// TIA Portal V20 export
DATA_BLOCK "ControlNodes"   // DB32
// stored: MemoryReserve 100, Namespace Unit1
   VAR
      em { ExternalWritable := 'False'} : "LAF_typeEmControlNode";
      fuse : Array[0..150] of Bool;
      pws : Array[0..10] of Bool;
      motorPowerMC { ExternalWritable := 'False'} : Struct
         FeedBack : Bool;
         mcOn : Bool;
         Ready : Bool;
         Operation : Bool;
         Run : Bool;
         Fault : Bool;
         Error : Bool;
      END_STRUCT;
      airOK { ExternalWritable := 'False'} : Bool;   // Compressed air OK
      InitializeEnable { ExternalWritable := 'False'} : Bool;
      AutoStartEnable { ExternalWritable := 'False'} : Bool;
      cmFFU_LIU117 : "LER_typeLIU117ControlNode";
      citiMap : "LER_OEM_Data";
      "========Communication========" : Bool;
      BA030 { ExternalWritable := 'False'} : "LER_typeCommunicationControlNode";
      BA040 { ExternalWritable := 'False'} : "LER_typeCommunicationControlNode";
      BA100 { S7_SetPoint := 'True'} : "LER_typeCommunicationControlNode";
      ConveyorA { ExternalWritable := 'False'} : "LER_typeCommunicationControlNode";
   END_VAR
BEGIN
   // fuse[0] : KISTLER 100KN PRESS POWER TRIPPED E202CB
   // fuse[1] : KISTLER 100KN PRESS POWER TRIPPED E208CB
   // fuse[2] : KISTLER 30KN PRESS POWER TRIPPED E214CB
   // fuse[3] : SPARE
   // fuse[4] : SPARE
   // fuse[5] : E8404PWS CONTROLLER POWER SMPS AC POWER TRIPPED E320CB
   // fuse[6] : E8704PWS SAFETY POWER SMPS AC POWER TRIPPED E326CB
   // fuse[7] : E8804PWS CONTRL POWER SMPS AC POWER TRIPPED E332CB
   // fuse[8] : PROCESSOR POWER ON TIPPRED E4120CB
   // fuse[9] : PROGRAMING POWER OUTLET TRPPED E4126CB
   // fuse[10] : SPARE
   // fuse[11] : PANEL LED POWER TRIPPED E4304CB
   // fuse[12] : SPARE
   // fuse[13] : CONTROL LEVEL HUB POWER TRIPPED E4420CB
   // fuse[14] : MAIN HMI POWER TRIPPED E4426CB
   // fuse[15] : PORTABLE HMI POWER TIPPED E4432CB
   // fuse[16] : PORTABLE HMI POWER TIPPED E4456CB
   // fuse[17] : 120VAC HEATER-1 POWER TR PRIMARY TRIPPED E5100CB
   // fuse[18] : SPARE
   // fuse[19] : SPARE
   // fuse[20] : UPPER 1-1 HEATER POWER TRIPPED E5156CB
   // fuse[21] : UPPER 1-2 HEATER POWER TRIPPED E5162CB
   // fuse[22] : LOWER 1-1 HEATER POWER TRIPPED E5168CB
   // fuse[23] : LOWER 1-2 HEATER POWER TRIPPED E5174CB
   // fuse[24] : LOWER 1-3 HEATER POWER TRIPPED E5180CB
   // fuse[25] : SPARE
   // fuse[26] : 120VAC HEATER-2 POWER TR PRIMARY TRIPPED E6100CB
   // fuse[27] : SPARE
   // fuse[28] : SPARE
   // fuse[29] : UPPER 2-1 HEATER POWER TRIPPED E6156CB
   // fuse[30] : UPPER 2-2 HEATER POWER TRIPPED E6162CB
   // fuse[31] : LOWER 2-1 HEATER POWER TRIPPED E6168CB
   // fuse[32] : LOWER 2-2 HEATER POWER TRIPPED E6174CB
   // fuse[33] : LOWER 2-3 HEATER POWER TRIPPED E6180CB
   // fuse[34] : SPARE
   // fuse[35] : 120VAC CONTROL POWER TR PRIMARY TRIPPED E7100CB
   // fuse[36] : 120VAC CONTROL POWER TR SECONDARY TRIPPED E7110CB
   // fuse[37] : CONTROL POWER ON TRIPPED E7116CB
   // fuse[38] : MOTOR PANEL CONTROL POWER TRIPPED E7154CB
   // fuse[39] : POWER STRIP OUTLET POWER TRIPPED E7160CB
   // fuse[40] : POWER STRIP OUTLET POWER TRIPPED E7166CB
   // fuse[41] : QR LASER MARKING TRIPPED E7172CB
   // fuse[42] : HI-POT TESTER POWER TRIPPED E7178CB
   // fuse[43] : FFU-1 POWER TRIPPED E7222CB
   // fuse[44] : UPPER 1-1 TEMPERATURE CONTROLLER POWER TRIPPED E5206CB
   // fuse[45] : UPPER 1-2 TEMPERATURE CONTROLLER POWER TRIPPED E5212CB
   // fuse[46] : LOWER 1-1 TEMPERATURE CONTROLLER POWER TRIPPED E5218CB
   // fuse[47] : LOWER 1-2 TEMPERATURE CONTROLLER POWER TRIPPED E5224CB
   // fuse[48] : LOWER 1-3 TEMPERATURE CONTROLLER POWER TRIPPED E5230CB
   // fuse[49] : UPPER 2-1 TEMPERATURE CONTROLLER POWER TRIPPED E6206CB
   // fuse[50] : UPPER 2-2 TEMPERATURE CONTROLLER POWER TRIPPED E6212CB
   // fuse[51] : LOWER 2-1 TEMPERATURE CONTROLLER POWER TRIPPED E6218CB
   // fuse[52] : LOWER 2-2 TEMPERATURE CONTROLLER POWER TRIPPED E6224CB
   // fuse[53] : LOWER 2-3 TEMPERATURE CONTROLLER POWER TRIPPED E6230CB
   // fuse[54] : SPARE
   // fuse[55] : ET200MP I/O OUTPUT POWER TRIPPED E8154CB
   // fuse[56] : JUNCTION BOX CONTROL POWER TRIPPED E8180CB
   // fuse[57] : CLASS 2 SMPS POWER TRIPPED E8204CB
   // fuse[58] : ET200ECO PN-1 POWER TRIPPED E8220CB
   // fuse[59] : ET200ECO PN-2 POWER TRIPPED E8224CB
   // fuse[60] : ET200ECO PN-3 POWER TRIPPED E8228CB
   // fuse[61] : ET200ECO PN-4 POWER TRIPPED E8232CB
   // fuse[62] : PANEL FAN POWER TRIPPED E8304CB
   // fuse[63] : SPARE
   // fuse[64] : CONTROLLER DC POWER TRIPPED E8406CB
   // fuse[65] : KISTLER CONTROL POWER TRIPPED E8416CB
   // fuse[66] : MANIFOLD-1 POWER TRIPPED E8422CB
   // fuse[67] : MANIFOLD-2 POWER TRIPPED E8430CB
   // fuse[68] : QR READER POWER TRIPPED E8456CB
   // fuse[69] : QR READER POWER TRIPPED E8462CB
   // fuse[70] : HANDY QR READER POWER TRIPPED E8468CB
   // fuse[71] : PROFINET CONVERTER POWER TRIPPED E8474CB
   // fuse[72] : MONITORING RELAY POWER TRIPPED E8504CB
   // fuse[73] : SPARE
   // fuse[74] : SAFETY DC POWER TRIPPED E8706CB
   // fuse[75] : ET200SP I/O SAFETY POWER TRIPPED E8716CB
   // fuse[76] : JUNCTION BOX CONTROL POWER TRIPPED E8736CB
   // fuse[77] : ET200ECO PN SAFETYT-1 POWER TRIPPED E8756CB
   // fuse[78] : ET200ECO PN SAFETYT-2 POWER TRIPPED E8762CB
   // fuse[79] : SPARE
   // fuse[80] : CONTROL DC POWER TRIPPED E8806CB
   // fuse[81] : JUNCTION BOX CONTROL POWER TRIPPED E8816CB
   // fuse[82] : DRIVE-CLIQ HUB POWER TRIPPED E8822CB
   // fuse[83] : EQUIPMENT LED POWER TRIPPED E8828CB
   // fuse[84] : SPARE
   // fuse[85] : SAFETY DC POWER TRIPPED E218CB
   // fuse[86] : CLASS 2 SMPS POWER TRIPPED E308CB
   // fuse[87] : ET200ECO PN-1 POWER TRIPPED E324CB
   // fuse[88] : ET200ECO PN-2 POWER TRIPPED E328CB
   // fuse[89] : ET200ECO PN-3 POWER TRIPPED E332CB
   // fuse[90] : ET200ECO PN-4 POWER TRIPPED E336CB
   // fuse[91] : MOTOR POWER MC FEEDBACK
   // fuse[92] : MOTOR POWER TRIPPED E202CB
   // fuse[93] : MAIN CONTROL PANEL MAIN POWER TRIPPED E208CB
   // fuse[94] : E6104PWS CONTROL POWER SMPS AC POWER TRIPPED E314CB
   // fuse[95] : JROUT P&P Y-AXIS POWER TR PRIMARY TRIPPED E400CB
   // fuse[96] : JROUT P&P Y-AXIS POWER TR ECONDARY TRIPPED E410CB
   // fuse[97] : INS PROCESS P&P X-AXIS POWER TR PRIMARY TRIPPED E500CB
   // fuse[98] : INS PROCESS P&P X-AXIS POWER TR ECONDARY TRIPPED E510CB
   // fuse[99] : JR UNLOADING Y-AXIS POWER TR PRIMARY TRIPPED E600CB
   // fuse[100] : JR UNLOADING Y-AXIS POWER TR ECONDARY TRIPPED E610CB
   // fuse[101] : POWER METER POWER TRIIPED E720CB
   // fuse[102] : POWER METER CONTROL POWER TRIIPED E726CB
   // fuse[103] : JR OUT P&P 1 Y-AXIS POWER ON TRIPPED E2004CB
   // fuse[104] : JR OUT P&P 2 Y-AXIS POWER ON TRIPPED E2104CB
   // fuse[105] : INS PROCESS P&P 1 X-AXIS POWER ON TRIPPED E2204CB
   // fuse[106] : INS PROCESS P&P 2 X-AXIS POWER ON TRIPPED E2304CB
   // fuse[107] : JR UNLOADING Y-AXIS POWER ON TRIPPED E2404CB
   // fuse[108] : MOTOR POWER MC COIL POWER TRIPPED E6156CB
   // fuse[109] : PROCESSOR POWER ON TRIPPRED E4116CB
   // fuse[110] : MAIN CONTROL PANEL HOT POWER TRIPPED E4156CB
   // fuse[111] : SYSTEM LEVEL HUB POWER TRIPPED E4162CB
   // fuse[112] : PANEL LED POWER TRIPPED E4304CB
   // fuse[113] : CONTROL POWER TRIPPED E5110CB
   // fuse[114] : CONTROL POWER ON TRIPPED E5120CB
   // fuse[115] : SERVON CONTROL POWER TRIPPED E6122CB
   // fuse[116] : SERVO CONTROL UNIT CONTROL POWER TRIPPED E6128CB
   // fuse[117] : PANEL FAN POWER TRIPPED E6204CB
   // fuse[118] : SPARE
   // fuse[119] : SPARE
   // fuse[120] : SPARE
   // fuse[121] : SPARE
   // pws[0] : PLC POWER SMPS DC OK E4404PWS
   // pws[1] : CONTROL POWER SMPS DC OK E8104PWS
   // pws[2] : CLASS 2 SMPS MONITORING E8206PWS
   // pws[3] : CONTROLLER POWER SMPS DC OK E8404PWS
   // pws[4] : SAFETY POWER SMPS DC OK E8704PWS
   // pws[5] : COONTRL POWER SMPS DC OK E8804PWS
   // pws[6] : CLASS 2 SMPS MONITORING E310PWS
   // pws[7] : CONTROL POWER SMPS DC OK E6104PWS
END_DATA_BLOCK
